	fbRPC:				ASyncRPC;
END_VAR


FunctionType:=FUNCTION_TYPE.FUNCTION_TYPE_ASYNC_RPC;
FunctionNumber:=GANTRY_ASYNC_FUNCTION_NUMBER.GANTRY_ASYNC_FUNCTION_PL;
ParameterDW:=0;
ParameterB:=0;
ParametersOK:=FALSE;

IF En THEN
	IF PickStation<=4 AND PickStation>=1 THEN
		IF PickPosition<=9 AND PickPosition>=1 THEN
			ParametersOK:=TRUE;
			ParameterDW:=INT_TO_DWORD((PickStation*1000+PickPosition*100) + (0*10+0));
		END_IF
	END_IF
END_IF

fbRPC(EN:=En AND ParametersOK, Data:=Data, FunctionType:=FunctionType,FunctionNumber:=FunctionNumber, ParameterDW:=ParameterDW, ParameterB:=ParameterB);

Done:=fbRPC.Done;
Executing:=fbRPC.Executing;
Waiting:=fbRPC.Waiting;
Error:=fbRPC.Error OR (fbRPC.Done AND fbRPC.ReturnValue<0) OR NOT ParametersOK;
Progress:=fbRPC.Progress;

END_FUNCTION_BLOCK

// ---- ComLib/POUs/Public/Level 6 Presentation/Gantry/GantryLeave.TcPOU
{library PUBLIC}
(*  Function to leave a pallet in a specific station and position.  *)
FUNCTION_BLOCK GantryLeave
VAR_INPUT
	En: 				BOOL:=FALSE;			(* Set to true to start *)
	LeaveStation:		StationType;			(* Station number 1-4 *)
	LeavePosition:		PositionType;			(* Position number 1-9 *)
END_VAR
VAR_OUTPUT
	Done: 				BOOL:=FALSE;			(* If true, the command is transmitted ok, to reset set En to false *)
	Executing:			BOOL:=FALSE;			(* True while the command in transmitted *)
	Waiting:			BOOL:=FALSE;			(* True if the command is queued to be transmitted *)
	Error: 				BOOL := FALSE;			(* True if an error occured *)
	Progress:			INT:=0;					(* Function progress *)
END_VAR
VAR_IN_OUT
	Data: 				CommunicationData;		(* Common data structure to connect this function block to a specific Communicator block *)
END_VAR
VAR
	FunctionType: 		FUNCTION_TYPE;
	FunctionNumber: 	INT;
	ParameterDW:	DWORD;
	ParameterB:		BYTE;
	ParametersOK:	BOOL;

	fbRPC:				ASyncRPC;
END_VAR


FunctionType:=FUNCTION_TYPE.FUNCTION_TYPE_ASYNC_RPC;
FunctionNumber:=GANTRY_ASYNC_FUNCTION_NUMBER.GANTRY_ASYNC_FUNCTION_PL;
ParameterDW:=0;
ParameterB:=0;
ParametersOK:=FALSE;

IF En THEN
	IF LeaveStation<=4 AND LeaveStation>=1 THEN
		IF LeavePosition<=9 AND LeavePosition>=1 THEN
			ParametersOK:=TRUE;
			ParameterDW:=INT_TO_DWORD( (0*1000+0*100) + (LeaveStation*10+LeavePosition));
		END_IF
	END_IF
END_IF

fbRPC(EN:=En AND ParametersOK, Data:=Data, FunctionType:=FunctionType,FunctionNumber:=FunctionNumber, ParameterDW:=ParameterDW, ParameterB:=ParameterB);

Done:=fbRPC.Done;
Executing:=fbRPC.Executing;
Waiting:=fbRPC.Waiting;
Error:=fbRPC.Error OR (fbRPC.Done AND fbRPC.ReturnValue<0) OR NOT ParametersOK;
Progress:=fbRPC.Progress;

END_FUNCTION_BLOCK

// ---- ComLib/POUs/Private/_FreeInstance.TcPOU
{library PRIVATE}
(*
  Private Funtcion:
  Frees a previous allocated communications instance.
  Note that it is not possible to free an instance during ongoing read or write (use cancel to break ongoing send or read).

  Return true if station was released. 
*)

FUNCTION _FreeInstance : BOOL
VAR_INPUT
	Instance: 				INT;		(* Instance, a number concatenated by SationNumber (1-INSTANCE_MAX_NUMBER_OF_STATIONS) and DeviceNumber (1-INSTANCE_MAX_NUMBER_OF_DEVICES). Instance is defined as: StaionNumber*100+DeviceNumber *)
END_VAR
VAR
	StationNumber: 		INT;
	StationDevice: 		INT;
END_VAR

_FreeInstance:=FALSE;

IF _CheckInstance(Instance) THEN
	StationNumber:=Instance/100;
	StationDevice:=Instance-StationNumber*100;

	IF ( ComGVL._Instance[StationNumber, StationDevice]<> INSTANCE_STATUS.INSTANCE_STATUS_BUSY) AND
              (ComGVL._Instance[StationNumber, StationDevice]<>INSTANCE_STATUS.INSTANCE_STATUS_CANCEL) THEN

		ComGVL._Instance[StationNumber, StationDevice]:=INSTANCE_STATUS.INSTANCE_STATUS_FREE;
		_FreeInstance:=TRUE;
	END_IF;
END_IF;

END_FUNCTION

// ---- ComLib/POUs/Private/_TryOut.TcPOU
{library PRIVATE}
FUNCTION_BLOCK _TryOut
VAR_INPUT
	Enable: BOOL;
END_VAR
VAR_OUTPUT
END_VAR
VAR
	ABBStatusRestart:		INT:=1;
	
END_VAR

ComGVL._fbTryOutShowABB:=FALSE;
ComGVL._fbTryOutShowGantry:=FALSE;

ComGVL._fbTryOutCommunicator(En:=ComGVL._mxTryOutEnable, Address:=ComGVL._miAddressNumber[ComGVL._miAddressIndex], Data:=ComGVL._msTryOutData);

CASE  ComGVL._glAddressSelectionIndex OF
1,2,3,4:
	ComGVL._fbTryOutShowABB:=TRUE;

	ComGVL._fbTryOutABBGetStatus(En:=ComGVL._fbTryOutABBGoToHomeEn, Data:=ComGVL._msTryOutData);
	IF ComGVL._fbTryOutABBGetStatus.Done THEN
		ComGVL._fbTryOutABBRunMode:=ComGVL._fbTryOutABBGetStatus.RunningMode;
		ComGVL._fbTryOutABBOpMode:=ComGVL._fbTryOutABBGetStatus.OperatingMode;
		ABBStatusRestart:=ABBStatusRestart+1;
		IF ABBStatusRestart=4 THEN
			ABBStatusRestart:=1;
			ComGVL._fbTryOutABBGetStatus(En:=FALSE, Data:=ComGVL._msTryOutData);
		END_IF;
	END_IF;

	(* GoTo *)
	ComGVL._fbTryOutABBGoToHome(En:=ComGVL._fbTryOutABBGoToHomeEn, Data:=ComGVL._msTryOutData);
	IF ComGVL._fbTryOutABBGoToHome.En THEN
		ComGVL._fbTryOutDone:=ComGVL._fbTryOutABBGoToHome.Done;
		ComGVL._fbTryOutExecuting:=ComGVL._fbTryOutABBGoToHome.Executing;
		ComGVL._fbTryOutWaiting:=ComGVL._fbTryOutABBGoToHome.Waiting;
		ComGVL._fbTryOutError:=ComGVL._fbTryOutABBGoToHome.Error;
		ComGVL._fbTryOutProgress:=ComGVL._fbTryOutABBGoToHome.Progress;
	END_IF;
	
	ComGVL._fbTryOutABBGoToSensor(En:=ComGVL._fbTryOutABBGoToSensorEn, Data:=ComGVL._msTryOutData);
	IF ComGVL._fbTryOutABBGoToSensor.En THEN
		ComGVL._fbTryOutDone:=ComGVL._fbTryOutABBGoToSensor.Done;
		ComGVL._fbTryOutExecuting:=ComGVL._fbTryOutABBGoToSensor.Executing;
		ComGVL._fbTryOutWaiting:=ComGVL._fbTryOutABBGoToSensor.Waiting;
		ComGVL._fbTryOutError:=ComGVL._fbTryOutABBGoToSensor.Error;
		ComGVL._fbTryOutProgress:=ComGVL._fbTryOutABBGoToSensor.Progress;
	END_IF;
	
	ComGVL._fbTryOutABBGoToStorage(En:=ComGVL._fbTryOutABBGoToStorageEn, Data:=ComGVL._msTryOutData);
	IF ComGVL._fbTryOutABBGoToStorage.En THEN
		ComGVL._fbTryOutDone:=ComGVL._fbTryOutABBGoToStorage.Done;
		ComGVL._fbTryOutExecuting:=ComGVL._fbTryOutABBGoToStorage.Executing;
		ComGVL._fbTryOutWaiting:=ComGVL._fbTryOutABBGoToStorage.Waiting;
		ComGVL._fbTryOutError:=ComGVL._fbTryOutABBGoToStorage.Error;
		ComGVL._fbTryOutProgress:=ComGVL._fbTryOutABBGoToStorage.Progress;
	END_IF;
	
	ComGVL._fbTryOutABBGoToTable(En:=ComGVL._fbTryOutABBGoToTableEn, Data:=ComGVL._msTryOutData);
	IF ComGVL._fbTryOutABBGoToTable.En THEN
		ComGVL._fbTryOutDone:=ComGVL._fbTryOutABBGoToTable.Done;
		ComGVL._fbTryOutExecuting:=ComGVL._fbTryOutABBGoToTable.Executing;
		ComGVL._fbTryOutWaiting:=ComGVL._fbTryOutABBGoToTable.Waiting;
		ComGVL._fbTryOutError:=ComGVL._fbTryOutABBGoToTable.Error;
		ComGVL._fbTryOutProgress:=ComGVL._fbTryOutABBGoToTable.Progress;
	END_IF;

	ComGVL._fbTryOutABBGoToConveyor1(En:=ComGVL._fbTryOutABBGoToConveyor1En, Data:=ComGVL._msTryOutData);
	IF ComGVL._fbTryOutABBGoToConveyor1.En THEN
		ComGVL._fbTryOutDone:=ComGVL._fbTryOutABBGoToConveyor1.Done;
		ComGVL._fbTryOutExecuting:=ComGVL._fbTryOutABBGoToConveyor1.Executing;
		ComGVL._fbTryOutWaiting:=ComGVL._fbTryOutABBGoToConveyor1.Waiting;
		ComGVL._fbTryOutError:=ComGVL._fbTryOutABBGoToConveyor1.Error;
		ComGVL._fbTryOutProgress:=ComGVL._fbTryOutABBGoToConveyor1.Progress;
	END_IF;
	
	ComGVL._fbTryOutABBGoToConveyor2(En:=ComGVL._fbTryOutABBGoToConveyor2En, Data:=ComGVL._msTryOutData);
	IF ComGVL._fbTryOutABBGoToConveyor2.En THEN
		ComGVL._fbTryOutDone:=ComGVL._fbTryOutABBGoToConveyor2.Done;
		ComGVL._fbTryOutExecuting:=ComGVL._fbTryOutABBGoToConveyor2.Executing;
		ComGVL._fbTryOutWaiting:=ComGVL._fbTryOutABBGoToConveyor2.Waiting;
		ComGVL._fbTryOutError:=ComGVL._fbTryOutABBGoToConveyor2.Error;
		ComGVL._fbTryOutProgress:=ComGVL._fbTryOutABBGoToConveyor2.Progress;
	END_IF;
	
	(* Pick Leave *)
	ComGVL._fbTryOutABBPickLeaveSensor(En:=ComGVL._fbTryOutABBPickLeaveSensorEn, Data:=ComGVL._msTryOutData, Pick:=ComGVL._fbTryOutABBPSensor);
	IF ComGVL._fbTryOutABBPickLeaveSensor.En THEN
		ComGVL._fbTryOutDone:=ComGVL._fbTryOutABBPickLeaveSensor.Done;
		ComGVL._fbTryOutExecuting:=ComGVL._fbTryOutABBPickLeaveSensor.Executing;
		ComGVL._fbTryOutWaiting:=ComGVL._fbTryOutABBPickLeaveSensor.Waiting;
		ComGVL._fbTryOutError:=ComGVL._fbTryOutABBPickLeaveSensor.Error;
		ComGVL._fbTryOutProgress:=ComGVL._fbTryOutABBPickLeaveSensor.Progress;
	END_IF;
	
	ComGVL._fbTryOutABBPickLeaveStorage(En:=ComGVL._fbTryOutABBPickLeaveStorageEn, Data:=ComGVL._msTryOutData, Pick:=ComGVL._fbTryOutABBPStorage, Position:=ComGVL._fbTryOutABBPStoragePos);
	IF ComGVL._fbTryOutABBPickLeaveStorage.En THEN
		ComGVL._fbTryOutDone:=ComGVL._fbTryOutABBPickLeaveStorage.Done;
		ComGVL._fbTryOutExecuting:=ComGVL._fbTryOutABBPickLeaveStorage.Executing;
		ComGVL._fbTryOutWaiting:=ComGVL._fbTryOutABBPickLeaveStorage.Waiting;
		ComGVL._fbTryOutError:=ComGVL._fbTryOutABBPickLeaveStorage.Error;
		ComGVL._fbTryOutProgress:=ComGVL._fbTryOutABBPickLeaveStorage.Progress;
	END_IF;
	
	ComGVL._fbTryOutABBPickLeaveTable(En:=ComGVL._fbTryOutABBPickLeaveTableEn, Data:=ComGVL._msTryOutData, Pick:=ComGVL._fbTryOutABBPTable, Position:=ComGVL._fbTryOutABBPTablePos);
	IF ComGVL._fbTryOutABBPickLeaveTable.En THEN
		ComGVL._fbTryOutDone:=ComGVL._fbTryOutABBPickLeaveTable.Done;
		ComGVL._fbTryOutExecuting:=ComGVL._fbTryOutABBPickLeaveTable.Executing;
		ComGVL._fbTryOutWaiting:=ComGVL._fbTryOutABBPickLeaveTable.Waiting;
		ComGVL._fbTryOutError:=ComGVL._fbTryOutABBPickLeaveTable.Error;
		ComGVL._fbTryOutProgress:=ComGVL._fbTryOutABBPickLeaveTable.Progress;
	END_IF;
	
	ComGVL._fbTryOutABBPickLeaveTable(En:=ComGVL._fbTryOutABBPickLeaveTableEn, Data:=ComGVL._msTryOutData, Pick:=ComGVL._fbTryOutABBPTable, Position:=ComGVL._fbTryOutABBPTablePos);
	IF ComGVL._fbTryOutABBPickLeaveTable.En THEN
		ComGVL._fbTryOutDone:=ComGVL._fbTryOutABBPickLeaveTable.Done;
		ComGVL._fbTryOutExecuting:=ComGVL._fbTryOutABBPickLeaveTable.Executing;
		ComGVL._fbTryOutWaiting:=ComGVL._fbTryOutABBPickLeaveTable.Waiting;
		ComGVL._fbTryOutError:=ComGVL._fbTryOutABBPickLeaveTable.Error;
		ComGVL._fbTryOutProgress:=ComGVL._fbTryOutABBPickLeaveTable.Progress;
	END_IF;
	
	ComGVL._fbTryOutABBPickLeaveConveyor1(En:=ComGVL._fbTryOutABBPickLeaveConveyor1En, Data:=ComGVL._msTryOutData, Pick:=ComGVL._fbTryOutABBPConveyor1);
	IF ComGVL._fbTryOutABBPickLeaveConveyor1.En THEN
		ComGVL._fbTryOutDone:=ComGVL._fbTryOutABBPickLeaveConveyor1.Done;
		ComGVL._fbTryOutExecuting:=ComGVL._fbTryOutABBPickLeaveConveyor1.Executing;
		ComGVL._fbTryOutWaiting:=ComGVL._fbTryOutABBPickLeaveConveyor1.Waiting;
		ComGVL._fbTryOutError:=ComGVL._fbTryOutABBPickLeaveConveyor1.Error;
		ComGVL._fbTryOutProgress:=ComGVL._fbTryOutABBPickLeaveConveyor1.Progress;
	END_IF;
	
	ComGVL._fbTryOutABBPickLeaveConveyor2(En:=ComGVL._fbTryOutABBPickLeaveConveyor2En, Data:=ComGVL._msTryOutData, Pick:=ComGVL._fbTryOutABBPConveyor2);
	IF ComGVL._fbTryOutABBPickLeaveConveyor2.En THEN
		ComGVL._fbTryOutDone:=ComGVL._fbTryOutABBPickLeaveConveyor2.Done;
		ComGVL._fbTryOutExecuting:=ComGVL._fbTryOutABBPickLeaveConveyor2.Executing;
		ComGVL._fbTryOutWaiting:=ComGVL._fbTryOutABBPickLeaveConveyor2.Waiting;
		ComGVL._fbTryOutError:=ComGVL._fbTryOutABBPickLeaveConveyor2.Error;
		ComGVL._fbTryOutProgress:=ComGVL._fbTryOutABBPickLeaveConveyor2.Progress;
	END_IF;

5:
	ComGVL._fbTryOutShowGantry:=TRUE;

	ComGVL._fbTryOutGantryPick(En:=ComGVL._fbTryOutGantryPickEn, Data:=ComGVL._msTryOutData, PickStation:=ComGVL._fbTryOutGantryPickStation, PickPosition:=ComGVL._fbTryOutGantryPickPos);
	IF ComGVL._fbTryOutGantryPick.En THEN
		ComGVL._fbTryOutDone:=ComGVL._fbTryOutGantryPick.Done;
		ComGVL._fbTryOutExecuting:=ComGVL._fbTryOutGantryPick.Executing;
		ComGVL._fbTryOutWaiting:=ComGVL._fbTryOutGantryPick.Waiting;
		ComGVL._fbTryOutError:=ComGVL._fbTryOutGantryPick.Error;
		ComGVL._fbTryOutProgress:=ComGVL._fbTryOutGantryPick.Progress;
	END_IF;

	ComGVL._fbTryOutGantryLeave(En:=ComGVL._fbTryOutGantryLeaveEn, Data:=ComGVL._msTryOutData, LeaveStation:=ComGVL._fbTryOutGantryLeaveStation, LeavePosition:=ComGVL._fbTryOutGantryLeavePos);
	IF ComGVL._fbTryOutGantryLeave.En THEN
		ComGVL._fbTryOutDone:=ComGVL._fbTryOutGantryLeave.Done;
		ComGVL._fbTryOutExecuting:=ComGVL._fbTryOutGantryLeave.Executing;
		ComGVL._fbTryOutWaiting:=ComGVL._fbTryOutGantryLeave.Waiting;
		ComGVL._fbTryOutError:=ComGVL._fbTryOutGantryLeave.Error;
		ComGVL._fbTryOutProgress:=ComGVL._fbTryOutGantryLeave.Progress;
	END_IF;

END_CASE

ComGVL._fbTryOutGetStatus(En:=TRUE, Data:=ComGVL._msTryOutData);
ComGVL._fbTryOutGetStatusRunning:=ComGVL._fbTryOutGetStatus.Running;
ComGVL._fbTryOutGetStatusProgress:=ComGVL._fbTryOutGetStatus.Progress;
ComGVL._fbTryOutGetStatusProgramNumber:=ComGVL._fbTryOutGetStatus.ProgramNumber;
ComGVL._fbTryOutGetStatusHeartBeat:=ComGVL._fbTryOutGetStatus.HeartBeat;
ComGVL._fbTryOutGetStatusError:=ComGVL._fbTryOutGetStatus.Error;

END_FUNCTION_BLOCK

// ---- ComLib/POUs/Public/Level 2 Data link/DeviceClose.TcPOU
{library PUBLIC}
(* Use this function to close an open communication link to a specific device defined by Instance.
Returnvalue is true if closed ok otherwise false.*)
FUNCTION DeviceClose : BOOL
VAR_INPUT
	Instance: 				INT;		(* Instance is an address, use the function ToAddress() to convert station and device number to a valid address. *)
END_VAR

DeviceClose:=FALSE;
IF _GetInstance(Instance)=INSTANCE_STATUS.INSTANCE_STATUS_READY THEN
	IF _FreeInstance(Instance) THEN
		DeviceClose:=TRUE;
	END_IF;
END_IF;

END_FUNCTION

// ---- ComLib/POUs/Public/Level 2 Data link/DeviceStatus.TcPOU
{library PUBLIC}
(* Use this function block toget status of a specific device instance.*)
FUNCTION_BLOCK DeviceStatus
VAR_INPUT
	En:						BOOL;		(* Enable signal, if true this block will give new status values *)
	Instance: 				INT;		(* Instance is an address, use the function ToAddress() to convert station and device number to a valid address. *)
END_VAR
VAR_OUTPUT
	Done:					BOOL:=FALSE;			(* True if status was read  *)
	Status: 				INSTANCE_STATUS;		(* Global status for a specific device *)
END_VAR
VAR
END_VAR

IF En THEN
	Status:=_GetInstance(Instance);
	Done:=TRUE;
ELSE
	Done:=FALSE;
END_IF;

END_FUNCTION_BLOCK

// ---- ComLib/POUs/Public/Level 2 Data link/DeviceUse.TcPOU
{library PUBLIC}
(* Use this function block to handle a communication link to a specific device defined by Instance.*)
FUNCTION_BLOCK DeviceUse
VAR_INPUT
	En:						BOOL;					(* Enable signal, if true this block will try to open the device  for communication use, if false and if device was opened it will be closed (Note: may take some time) *)
	Instance: 				INT;					(* Instance is an address, use the function ToAddress() to convert station and device number to a valid address. *)
END_VAR
VAR_OUTPUT
	Done:					BOOL:=FALSE;		(* True if a device was open (note: will remain false until a device is open), will go to false when a previous open device is closed *)
	Status: 				INSTANCE_STATUS;	(* Global status for a specific device *)
END_VAR
VAR
	OldInstance: INT;
END_VAR

Status:=_GetInstance(Instance);

IF En THEN
	IF Status=INSTANCE_STATUS.INSTANCE_STATUS_FREE THEN
		Done:=DeviceOpen(Instance);
		OldInstance:=Instance;
	END_IF;
ELSE
	IF Done THEN
		IF DeviceClose(OldInstance) THEN
			Done:=FALSE;
		END_IF;
	END_IF;
END_IF;

END_FUNCTION_BLOCK

// ---- ComLib/POUs/Public/Level 5 Session/RPC Remote Procedural Call/ASyncProgress.TcPOU
{library PUBLIC}
(*
Get progress value for ASync calls.
This function block will read the global status.
To see a specific function progress use the output of RPCx or ASyncRP function blocks.
*)

FUNCTION_BLOCK ASyncProgress
VAR_INPUT
	En: 				BOOL;			(* Set to true to get progress value *)
END_VAR
VAR_OUTPUT
	Done:				BOOL;			(* Done = En *)
	Progress: 			INT;			(* Progress value *)
END_VAR
VAR_IN_OUT
	Data: 				CommunicationData;		(* Common data structure to connect this function block to a specific Communicator block *)
END_VAR
VAR
END_VAR

IF En THEN
	Progress:=Data._ASyncProgress;
ELSE
	Progress:=0;
END_IF;

Done:=En;

END_FUNCTION_BLOCK

// ---- ComLib/POUs/Public/Level 5 Session/RPC Remote Procedural Call/RPC2.TcPOU
{library PUBLIC}
(*
RPC2 will handle RPC calls with 2 parameters.
A session will be established to the specific equipment during the function call and when a return value exist (or error) the session is ended.
Note, if FunctionType is set to ASync, RPC will only start a function and not wait for the function to end.

It is possible to queue many calls by cascade coupled blocks in serie or parallel.
By using the Done output signal as input to En on another function blockit is possible to serialise calls.

*)
FUNCTION_BLOCK RPC2
VAR_INPUT
	En: 				BOOL:=FALSE;			(* Set to true to call a  RPC 1 parameter function *)
	FunctionType1:	FUNCTION_TYPE:=FUNCTION_TYPE.FUNCTION_TYPE_SYNC_RPC;		(* Function type 1 must be of type SYNC *)
	FunctionNumber1:INT;						(* RPC function number 1 *)
	ParameterDW1:	DWORD;					(* DWORD parameter value 1 *)
	ParameterB1:		BYTE;						(* Byte parameter value 1 *)
	FunctionType2:	FUNCTION_TYPE:=FUNCTION_TYPE.FUNCTION_TYPE_SYNC_RPC;		(*Function type 2 must be of type SYNC *)
	FunctionNumber2:INT;						(* RPC function number 2 *)
	ParameterDW2:	DWORD;					(* DWORD parameter value 2 *)
	ParameterB2:		BYTE;						(* Byte parameter value 2 *)
END_VAR
VAR_OUTPUT
	Done: 				BOOL:=FALSE;			(* If true, the command is transmitted ok, to reset set En to false *)
	Executing:			BOOL:=FALSE;			(* True while the command in transmitted *)
	Waiting:			BOOL:=FALSE;			(* True if the command is queued to be transmitted *)
	Error: 				BOOL := FALSE;			(* True if an communication error occured *)
	ReturnValue1:		FUNCTION_TYPE;		(* Return value *)
	ReturnValue2:		DWORD;					(* DWORD return value *)
	ReturnValue3:		BYTE;						(* BYTE return value *)
END_VAR
VAR_IN_OUT
	Data: 				CommunicationData;		(* Common data structure to connect this function block to a specific Communicator block *)
END_VAR
VAR
	fbSessionInit: 		SessionInit;
	fbSessionSend1: 	SessionSend;
	fbSessionSend2: 	SessionSend;
	fbSessionEnd: 	SessionEnd;
	Memory: 			BOOL := FALSE;
END_VAR

fbSessionInit(En:=En, Data:=Data);
fbSessionSend1(En:=fbSessionInit.Done, SessionID:=fbSessionInit.SessionID, Data:=Data,
					FunctionType:=INT_TO_BYTE(FunctionType1), FunctionNumber:=INT_TO_BYTE(FunctionNumber1),
 					ParameterDW:=ParameterDW1, ParameterB:=ParameterB1);

fbSessionSend2(En:=fbSessionInit.Done, SessionID:=fbSessionInit.SessionID, Data:=Data,
					FunctionType:=INT_TO_BYTE(FunctionType2), FunctionNumber:=INT_TO_BYTE(FunctionNumber2),
					ParameterDW:=ParameterDW2, ParameterB:=ParameterB2);

fbSessionEnd(En:=fbSessionSend2.Done, Data:=Data);

Done:=fbSessionSend2.Done;
Executing:=fbSessionSend1.Executing OR fbSessionSend1.Executing;
Waiting:=fbSessionSend1.Waiting;
Error:=fbSessionSend1.Error OR fbSessionSend2.Error;


IF fbSessionSend2.Done AND NOT Memory THEN
	Memory:=TRUE;
	ReturnValue1:=fbSessionSend2.Answer.FunctionType;
	ReturnValue2:=fbSessionSend2.Answer.ParameterDW;
	ReturnValue3:=fbSessionSend2.Answer.ParameterB;
ELSIF NOT En THEN
	ReturnValue1:=FUNCTION_TYPE.FUNCTION_TYPE_ERROR_NO_FUNCTION;
	Memory:=FALSE;
ELSE
	Memory:=FALSE;
	ReturnValue1:=FUNCTION_TYPE.FUNCTION_TYPE_ERROR_BUSY;
END_IF;

END_FUNCTION_BLOCK

// ---- ComLib/POUs/Public/Level 6 Presentation/ABB/IO/ABBIORead.TcPOU
{library PUBLIC}
(* Function to read a DI I/O *)
FUNCTION_BLOCK ABBIORead
VAR_INPUT
	En: 			BOOL:=FALSE;				(* Set to true to start *)
	IONumber:		INT:=0;						(* DI I/O number to read *)
END_VAR
VAR_OUTPUT
	Done: 				BOOL:=FALSE;			(* If true, the command is transmitted ok, to reset set En to false *)
	Executing:			BOOL:=FALSE;			(* True while the command in transmitted *)
	Waiting:			BOOL:=FALSE;			(* True if the command is queued to be transmitted *)
	Error: 				BOOL := FALSE;			(* True if an error occured *)
	Progress:			INT:=0;					(* Function progress *)
	Value:				BOOL:=FALSE;			(* I/O return value *)
END_VAR
VAR_IN_OUT
	Data: 				CommunicationData;		(* Common data structure to connect this function block to a specific Communicator block *)
END_VAR
VAR
	FunctionType: 		FUNCTION_TYPE;
	FunctionNumber: 	INT;
	ParameterDW:		DWORD;
	ParameterB:			BYTE;
	Sequence:			INT:=0;

	fbRPC:				RPC1;
END_VAR

FunctionType:=FUNCTION_TYPE.FUNCTION_TYPE_SYNC_RPC;
FunctionNumber:=ABB_SYNC_FUNCTION_NUMBER.ABB_SYNC_READ_DI;
ParameterDW:=INT_TO_DWORD(IONumber);

fbRPC(EN:=En, Data:=Data, FunctionType1:=FunctionType,FunctionNumber1:=FunctionNumber, ParameterDW1:=ParameterDW, ParameterB1:=ParameterB);

Done:=fbRPC.Done;
Executing:=fbRPC.Executing;
Waiting:=fbRPC.Waiting;
Error:=fbRPC.Error;
Progress:=100*BOOL_TO_INT(Done);
Value:=BYTE_TO_BOOL(fbRPC.ReturnValue3);

END_FUNCTION_BLOCK

// ---- ComLib/POUs/Public/Level 6 Presentation/ABB/IO/ABBIOReadValve.TcPOU
{library PUBLIC}
(* Function to read a valve value (open or closed) *)
FUNCTION_BLOCK ABBIOReadValve
VAR_INPUT
	En: 			BOOL:=FALSE;				(* Set to true to start *)
	Valve:			INT:=0;						(* Valve I/O number *)
END_VAR
VAR_OUTPUT
	Done: 				BOOL:=FALSE;			(* If true, the command is transmitted ok, to reset set En to false *)
	Executing:			BOOL:=FALSE;			(* True while the command in transmitted *)
	Waiting:			BOOL:=FALSE;			(* True if the command is queued to be transmitted *)
	Error: 				BOOL := FALSE;			(* True if an error occured *)
	Progress:			INT:=0;					(* Function progress *)
	Value:				BOOL:=FALSE;			(* FALSE=open, TRUE=closed *)
END_VAR
VAR_IN_OUT
	Data: 				CommunicationData;		(* Common data structure to connect this function block to a specific Communicator block *)
END_VAR
VAR
	FunctionType: 		FUNCTION_TYPE;
	FunctionNumber: 	INT;
	ParameterDW:	DWORD;
	ParameterB:		BYTE;
	Sequence:			INT:=0;

	fbRPC:				RPC1;
END_VAR

FunctionType:=FUNCTION_TYPE.FUNCTION_TYPE_SYNC_RPC;
FunctionNumber:=ABB_SYNC_FUNCTION_NUMBER.ABB_SYNC_WRITE_DO;
ParameterDW:=INT_TO_DWORD(Valve);
ParameterB:=0;

fbRPC(EN:=En, Data:=Data, FunctionType1:=FunctionType,FunctionNumber1:=FunctionNumber, ParameterDW1:=ParameterDW, ParameterB1:=ParameterB);

Done:=fbRPC.Done;
Executing:=fbRPC.Executing;
Waiting:=fbRPC.Waiting;
Error:=fbRPC.Error;
Progress:=100*BOOL_TO_INT(Done);
Value:=BYTE_TO_BOOL(fbRPC.ReturnValue3);

END_FUNCTION_BLOCK

// ---- ComLib/POUs/Public/Level 6 Presentation/ABB/IO/ABBIOWrite.TcPOU
{library PUBLIC}
(* Function to write a DO I/O *)
FUNCTION_BLOCK ABBIOWrite
VAR_INPUT
	En: 			BOOL:=FALSE;				(* Set to true to start *)
	IONumber:		INT:=0;						(* DO I/O number to read *)
END_VAR
VAR_OUTPUT
	Done: 				BOOL:=FALSE;			(* If true, the command is transmitted ok, to reset set En to false *)
	Executing:			BOOL:=FALSE;			(* True while the command in transmitted *)
	Waiting:			BOOL:=FALSE;			(* True if the command is queued to be transmitted *)
	Error: 				BOOL := FALSE;			(* True if an error occured *)
	Progress:			INT:=0;					(* Function progress *)
END_VAR
VAR_IN_OUT
	Data: 				CommunicationData;		(* Common data structure to connect this function block to a specific Communicator block *)
END_VAR
VAR
	FunctionType: 		FUNCTION_TYPE;
	FunctionNumber: 	INT;
	ParameterDW:	DWORD;
	ParameterB:		BYTE;
	Sequence:			INT:=0;

	fbRPC:				RPC1;
END_VAR

FunctionType:=FUNCTION_TYPE.FUNCTION_TYPE_SYNC_RPC;
FunctionNumber:=ABB_SYNC_FUNCTION_NUMBER.ABB_SYNC_WRITE_DO;
ParameterDW:=INT_TO_DWORD(IONumber);

fbRPC(EN:=En, Data:=Data, FunctionType1:=FunctionType,FunctionNumber1:=FunctionNumber, ParameterDW1:=ParameterDW, ParameterB1:=ParameterB);

Done:=fbRPC.Done;
Executing:=fbRPC.Executing;
Waiting:=fbRPC.Waiting;
Error:=fbRPC.Error;
Progress:=100*BOOL_TO_INT(Done);

END_FUNCTION_BLOCK

// ---- ComLib/POUs/Public/Level 6 Presentation/ABB/IO/ABBIOWriteValve.TcPOU
{library PUBLIC}
(* Function to write a value to valve I/O *)
FUNCTION_BLOCK ABBIOWriteValve
VAR_INPUT
	En: 			BOOL:=FALSE;				(* Set to true to start *)
	Valve:			INT:=0;							(* Valve I/O number *)
	Value:			BOOL:=FALSE;				(* FALSE=open, TRUE=closed *)
END_VAR
VAR_OUTPUT
	Done: 				BOOL:=FALSE;			(* If true, the command is transmitted ok, to reset set En to false *)
	Executing:			BOOL:=FALSE;			(* True while the command in transmitted *)
	Waiting:			BOOL:=FALSE;			(* True if the command is queued to be transmitted *)
	Error: 				BOOL := FALSE;			(* True if an error occured *)
	Progress:			INT:=0;					(* Function progress *)
END_VAR
VAR_IN_OUT
	Data: 				CommunicationData;		(* Common data structure to connect this function block to a specific Communicator block *)
END_VAR
VAR
	FunctionType: 		FUNCTION_TYPE;
	FunctionNumber: 	INT;
	ParameterDW:	DWORD;
	ParameterB:		BYTE;
	Sequence:			INT:=0;

	fbRPC:				RPC1;
END_VAR

FunctionType:=FUNCTION_TYPE.FUNCTION_TYPE_SYNC_RPC;
FunctionNumber:=ABB_SYNC_FUNCTION_NUMBER.ABB_SYNC_WRITE_DO;
ParameterDW:=INT_TO_DWORD(Valve);
ParameterB:=BOOL_TO_BYTE(Value);

fbRPC(EN:=En, Data:=Data, FunctionType1:=FunctionType,FunctionNumber1:=FunctionNumber, ParameterDW1:=ParameterDW, ParameterB1:=ParameterB);

Done:=fbRPC.Done;
Executing:=fbRPC.Executing;
Waiting:=fbRPC.Waiting;
Error:=fbRPC.Error;
Progress:=100*BOOL_TO_INT(Done);

END_FUNCTION_BLOCK

// ---- ComLib/POUs/Public/Level 6 Presentation/ABB/Move/ABBMoveJAbs.TcPOU
{library PUBLIC}
(* Function to move a robot to an abs location *)
FUNCTION_BLOCK ABBMoveJAbs
VAR_INPUT
	En: 				BOOL:=FALSE;			(* Set to true to start *)
	X:					REAL:=0.0;				(* X position *)
	Y:					REAL:=0.0;				(* Y position *)
	Z:					REAL:=0.0;				(* Z position *)
	RX:					REAL:=0.0;				(* RX angle *)
	RY:					REAL:=0.0;				(* RY angle *)
	RZ:					REAL:=0.0;				(* RZ angle *)
END_VAR
VAR_OUTPUT
	Done: 				BOOL:=FALSE;			(* If true, the command is transmitted ok, to reset set En to false *)
	Executing:			BOOL:=FALSE;			(* True while the command in transmitted *)
	Waiting:			BOOL:=FALSE;			(* True if the command is queued to be transmitted *)
	Error: 				BOOL := FALSE;			(* True if an error occured *)
	Progress:			INT:=0;					(* Function progress *)
END_VAR
VAR_IN_OUT
	Data: 				CommunicationData;		(* Common data structure to connect this function block to a specific Communicator block *)
END_VAR
VAR
	FunctionType: 		FUNCTION_TYPE;
	FunctionNumber: 	INT;
	ParameterDW:	DWORD;
	ParameterB:		BYTE;
	Sequence:			INT:=0;

	fbRPC:				ASyncRPC;
END_VAR

FunctionType:=FUNCTION_TYPE.FUNCTION_TYPE_ASYNC_RPC;
FunctionNumber:=ABB_ASYNC_ABS_MOVEJ_TO_POSE;
ParameterDW:=0;										(* No parameters *)
ParameterB:=0;

fbRPC(EN:=En, Data:=Data, FunctionType:=FunctionType,FunctionNumber:=FunctionNumber, ParameterDW:=ParameterDW, ParameterB:=ParameterB);

Done:=fbRPC.Done;
Executing:=fbRPC.Executing;
Waiting:=fbRPC.Waiting;
Error:=fbRPC.Error OR (fbRPC.Done AND fbRPC.ReturnValue<0);
Progress:=fbRPC.Progress;

END_FUNCTION_BLOCK

// ---- ComLib/POUs/Public/Level 6 Presentation/ABB/Move/ABBMoveJRel.TcPOU
{library PUBLIC}
(* Function to move a robot relative current location *)
FUNCTION_BLOCK ABBMoveJRel
VAR_INPUT
	En: 				BOOL:=FALSE;			(* Set to true to start *)
	X:					REAL:=0.0;				(* X position *)
	Y:					REAL:=0.0;				(* Y position *)
	Z:					REAL:=0.0;				(* Z position *)
	RX:					REAL:=0.0;				(* RX angle *)
	RY:					REAL:=0.0;				(* RY angle *)
	RZ:					REAL:=0.0;				(* RZ angle *)
END_VAR
VAR_OUTPUT
	Done: 				BOOL:=FALSE;			(* If true, the command is transmitted ok, to reset set En to false *)
	Executing:			BOOL:=FALSE;			(* True while the command in transmitted *)
	Waiting:			BOOL:=FALSE;			(* True if the command is queued to be transmitted *)
	Error: 				BOOL := FALSE;			(* True if an error occured *)
	Progress:			INT:=0;						(* Function progress *)
END_VAR
VAR_IN_OUT
	Data: 				CommunicationData;		(* Common data structure to connect this function block to a specific Communicator block *)
END_VAR
VAR
	FunctionType: 		FUNCTION_TYPE;
	FunctionNumber: 	INT;
	ParameterDW:	DWORD;
	ParameterB:		BYTE;
	Sequence:			INT:=0;

	fbRPC:				ASyncRPC;
END_VAR

FunctionType:=FUNCTION_TYPE.FUNCTION_TYPE_ASYNC_RPC;
FunctionNumber:=ABB_ASYNC_REL_MOVEJ_TO_POSE;
ParameterDW:=0;										(* No parameters *)
ParameterB:=0;

fbRPC(EN:=En, Data:=Data, FunctionType:=FunctionType,FunctionNumber:=FunctionNumber, ParameterDW:=ParameterDW, ParameterB:=ParameterB);

Done:=fbRPC.Done;
Executing:=fbRPC.Executing;
Waiting:=fbRPC.Waiting;
Error:=fbRPC.Error OR (fbRPC.Done AND fbRPC.ReturnValue<0);
Progress:=fbRPC.Progress;

END_FUNCTION_BLOCK

// ---- ComLib/POUs/Public/Level 6 Presentation/ABB/Move/ABBMoveLAbs.TcPOU
{library PUBLIC}
(* Function to move a robot to an abs location *)
FUNCTION_BLOCK ABBMoveLAbs
VAR_INPUT
	En: 				BOOL:=FALSE;			(* Set to true to start *)
	X:					REAL:=0.0;				(* X position *)
	Y:					REAL:=0.0;				(* Y position *)
	Z:					REAL:=0.0;				(* Z position *)
	RX:					REAL:=0.0;				(* RX angle *)
	RY:					REAL:=0.0;				(* RY angle *)
	RZ:					REAL:=0.0;				(* RZ angle *)
END_VAR
VAR_OUTPUT
	Done: 				BOOL:=FALSE;			(* If true, the command is transmitted ok, to reset set En to false *)
	Executing:			BOOL:=FALSE;			(* True while the command in transmitted *)
	Waiting:			BOOL:=FALSE;			(* True if the command is queued to be transmitted *)
	Error: 				BOOL := FALSE;			(* True if an error occured *)
	Progress:			INT:=0;						(* Function progress *)
END_VAR
VAR_IN_OUT
	Data: 				CommunicationData;		(* Common data structure to connect this function block to a specific Communicator block *)
END_VAR
VAR
	FunctionType: 		FUNCTION_TYPE;
	FunctionNumber: 	INT;
	ParameterDW:	DWORD;
	ParameterB:		BYTE;
	Sequence:			INT:=0;

	fbRPC:				ASyncRPC;
END_VAR

FunctionType:=FUNCTION_TYPE.FUNCTION_TYPE_ASYNC_RPC;
FunctionNumber:=ABB_ASYNC_ABS_MOVEL_TO_POSE;
ParameterDW:=0;										(* No parameters *)
ParameterB:=0;

fbRPC(EN:=En, Data:=Data, FunctionType:=FunctionType,FunctionNumber:=FunctionNumber, ParameterDW:=ParameterDW, ParameterB:=ParameterB);

Done:=fbRPC.Done;
Executing:=fbRPC.Executing;
Waiting:=fbRPC.Waiting;
Error:=fbRPC.Error OR (fbRPC.Done AND fbRPC.ReturnValue<0);
Progress:=fbRPC.Progress;

END_FUNCTION_BLOCK

// ---- ComLib/POUs/Public/Level 6 Presentation/ABB/Move/ABBMoveLRel.TcPOU
{library PUBLIC}
(* Function to move a robot relative current location *)
FUNCTION_BLOCK ABBMoveLRel
VAR_INPUT
	En: 				BOOL:=FALSE;			(* Set to true to start *)
	X:					REAL:=0.0;				(* X position *)
	Y:					REAL:=0.0;				(* Y position *)
	Z:					REAL:=0.0;				(* Z position *)
	RX:					REAL:=0.0;				(* RX angle *)
	RY:					REAL:=0.0;				(* RY angle *)
	RZ:					REAL:=0.0;				(* RZ angle *)
END_VAR
VAR_OUTPUT
	Done: 				BOOL:=FALSE;			(* If true, the command is transmitted ok, to reset set En to false *)
	Executing:			BOOL:=FALSE;			(* True while the command in transmitted *)
	Waiting:			BOOL:=FALSE;			(* True if the command is queued to be transmitted *)
	Error: 				BOOL := FALSE;			(* True if an error occured *)
	Progress:			INT:=0;						(* Function progress *)
END_VAR
VAR_IN_OUT
	Data: 				CommunicationData;		(* Common data structure to connect this function block to a specific Communicator block *)
END_VAR
VAR
	FunctionType: 		FUNCTION_TYPE;
	FunctionNumber: 	INT;
	ParameterDW:	DWORD;
	ParameterB:		BYTE;
	Sequence:			INT:=0;

	fbRPC:				ASyncRPC;
END_VAR

FunctionType:=FUNCTION_TYPE.FUNCTION_TYPE_ASYNC_RPC;
FunctionNumber:=ABB_ASYNC_REL_MOVEL_TO_POSE;
ParameterDW:=0;										(* No parameters *)
ParameterB:=0;

fbRPC(EN:=En, Data:=Data, FunctionType:=FunctionType,FunctionNumber:=FunctionNumber, ParameterDW:=ParameterDW, ParameterB:=ParameterB);

Done:=fbRPC.Done;
Executing:=fbRPC.Executing;
Waiting:=fbRPC.Waiting;
Error:=fbRPC.Error OR (fbRPC.Done AND fbRPC.ReturnValue<0);
Progress:=fbRPC.Progress;

END_FUNCTION_BLOCK

// ---- ComLib/POUs/Public/Level 6 Presentation/ABB/Pick Leave/ABBProcessAssembly.TcPOU
{library PUBLIC}
(* Function to start a assembly process on the table. *)
FUNCTION_BLOCK ABBProcessAssembly
VAR_INPUT
	En: 				BOOL:=FALSE;			(* Set to true to start *)
END_VAR
VAR_OUTPUT
	Done: 				BOOL:=FALSE;			(* If true, the command is transmitted ok, to reset set En to false *)
	Executing:			BOOL:=FALSE;			(* True while the command in transmitted *)
	Waiting:			BOOL:=FALSE;			(* True if the command is queued to be transmitted *)
	Error: 				BOOL := FALSE;			(* True if an error occured *)
	Progress:			INT:=0;						(* Function progress *)
END_VAR
VAR_IN_OUT
	Data: 				CommunicationData;		(* Common data structure to connect this function block to a specific Communicator block *)
END_VAR
VAR
	FunctionType: 		FUNCTION_TYPE;
	FunctionNumber: 	INT;
	ParameterDW:	DWORD;
	ParameterB:		BYTE;
	Sequence:			INT:=0;

	fbRPC:				ASyncRPC;
END_VAR

FunctionType:=FUNCTION_TYPE.FUNCTION_TYPE_ASYNC_RPC;
FunctionNumber:=ABB_ASYNC_FUNCTION_PROCESS_ASSEMBLY;
ParameterDW:=0;
ParameterB:=0;

fbRPC(EN:=En, Data:=Data, FunctionType:=FunctionType,FunctionNumber:=FunctionNumber, ParameterDW:=ParameterDW, ParameterB:=ParameterB);

Done:=fbRPC.Done;
Executing:=fbRPC.Executing;
Waiting:=fbRPC.Waiting;
Error:=fbRPC.Error OR (fbRPC.Done AND fbRPC.ReturnValue<0);
Progress:=fbRPC.Progress;

END_FUNCTION_BLOCK

// ---- ComLib/POUs/Public/Level 6 Presentation/Gantry/GantryStatus.TcPOU
{library PUBLIC}
(* Function to get gantry status.
    This function can run continuously and will not block other communications.   
 *)
FUNCTION_BLOCK GantryStatus
VAR_INPUT
	En: 					BOOL:=FALSE;			(* Set to true to ask for status, the block  will continuously ask for status while true *)
END_VAR
VAR_OUTPUT
	Done: 					BOOL:=FALSE;			(* If true, the STATUS command is running, to stop/pause set En to false *)
	Status:					GANTRY_STATUS;			(* Gantry status *)
END_VAR
VAR_IN_OUT
	Data: 					CommunicationData;		(* Common data structure to connect this function block to a specific Communicator block *)
END_VAR
VAR
END_VAR


IF En THEN
	
	Status:=NodeReadWord(Address:=Data._Address, Channel:=2);
	Done:=TRUE;
ELSE
	Status:=GANTRY_STATUS.GANTRY_STATUS_NOT_ENABLED;
	Done:=FALSE;
END_IF;

END_FUNCTION_BLOCK

// ---- ComLib/VISUs/Object/_VisuABBGoTo.TcVIS
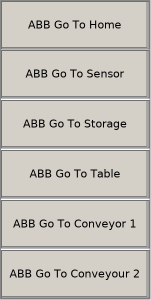
VISUALIZATION _VisuABBGoTo  // 151x300
    Button (1,1 148x48), "ABB Go To Home"
        toggle ComGVL._fbTryOutABBGoToHomeEn
    Button (1,50 148x48), "ABB Go To Sensor"
        toggle ComGVL._fbTryOutABBGoToSensorEn
    Button (1,100 148x48), "ABB Go To Storage"
        toggle ComGVL._fbTryOutABBGoToStorageEn
    Button (1,150 148x48), "ABB Go To Table"
        toggle ComGVL._fbTryOutABBGoToTableEn
    Button (1,200 148x48), "ABB Go To Conveyor 1"
        toggle ComGVL._fbTryOutABBGoToConveyor1En
    Button (1,250 148x48), "ABB Go To Conveyour 2"
        toggle ComGVL._fbTryOutABBGoToConveyor2En
END_VISUALIZATION

// ---- ComLib/VISUs/Object/_VisuABBPickLeave.TcVIS
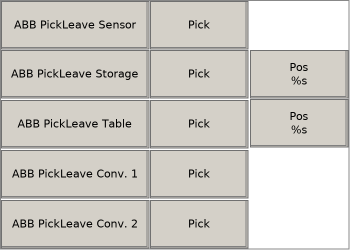
VISUALIZATION _VisuABBPickLeave  // 350x250
    Button (1,1 148x48), "ABB PickLeave Sensor"
        toggle ComGVL._fbTryOutABBPickLeaveSensorEn
    Button (1,50 148x48), "ABB PickLeave Storage"
        toggle ComGVL._fbTryOutABBPickLeaveStorageEn
    Button (1,100 148x48), "ABB PickLeave Table"
        toggle ComGVL._fbTryOutABBPickLeaveTableEn
    Button (1,150 148x48), "ABB PickLeave Conv. 1"
        toggle ComGVL._fbTryOutABBPickLeaveConveyor1En
    Button (1,200 148x48), "ABB PickLeave Conv. 2"
        toggle ComGVL._fbTryOutABBPickLeaveConveyor2En
    Button (150,1 98x48), "Pick"
        toggle ComGVL._fbTryOutABBPSensor
    Button (150,50 98x48), "Pick"
        toggle ComGVL._fbTryOutABBPStorage
    Button (150,100 98x48), "Pick"
        toggle ComGVL._fbTryOutABBPTable
    Button (150,150 98x48), "Pick"
        toggle ComGVL._fbTryOutABBPConveyor1
    Button (150,200 98x48), "Pick"
        toggle ComGVL._fbTryOutABBPConveyor2
    Button (250,50 98x48), "Pos %s", text variable: ComGVL._fbTryOutABBPStoragePos
        OnMouseClick: write the text variable via VisuDialogs.Numpad, min 1, max 9, title 'Position'
    Button (250,99 98x48), "Pos %s", text variable: ComGVL._fbTryOutABBPTablePos
        OnMouseClick: write the text variable via VisuDialogs.Numpad, min 1, max 9, title 'Position'
END_VISUALIZATION

// ---- ComLib/VISUs/Object/_VisuABBStatus.TcVIS
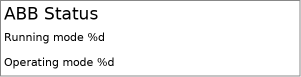
VISUALIZATION _VisuABBStatus  // 301x77
    Label (1,1 148x25), "ABB Status"
    Rectangle (1,25 298x25), "Running mode %d", text variable: ComGVL._gABBRunTable[ComGVL._fbTryOutABBRunMode ]
    Rectangle (1,50 298x25), "Operating mode %d", text variable: ComGVL._gABBOpTable[ComGVL._fbTryOutABBOpMode ]
END_VISUALIZATION

// ---- ComLib/VISUs/Object/_VisuAddressSelector.TcVIS
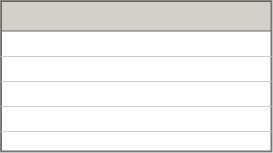
VISUALIZATION _VisuAddressSelector  // 273x153
    Table (1,1 270x150), data array: ComGVL._glAddressNameTable
        p3854506369: ComGVL._glAddressNameTable[INDEX]
        p2232123230: Station Address
        p1137915858: ComGVL._glAddressSelectionIndex
END_VISUALIZATION

// ---- ComLib/VISUs/Object/_VisuAddressShow.TcVIS
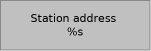
VISUALIZATION _VisuAddressShow  // 151x51
    Rectangle (1,1 148x48), "Station address %s", text variable: ComGVL._glAddressNameTable[ComGVL._glAddressSelectionIndex]
END_VISUALIZATION

// ---- ComLib/VISUs/Object/_VisuCommunicator.TcVIS
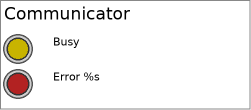
VISUALIZATION _VisuCommunicator  // 251x110
    Lamp1 (1,25 34x48), variable: ComGVL._fbTryOutCommunicator.Busy, style: Lamp-Lamp1-Yellow
    Rectangle (50,25 100x34), "Busy"
    Label (1,1 248x25), "Communicator"
    Lamp1 (1,60 34x48), variable: ComGVL._fbTryOutCommunicator.Error, style: Lamp-Lamp1-Red
    Rectangle (50,60 100x34), "Error %s", text variable: ComGVL._glErrorTable[ComGVL._fbTryOutCommunicator.ErrorID]
END_VISUALIZATION

// ---- ComLib/VISUs/Object/_VisuFunctionCall.TcVIS
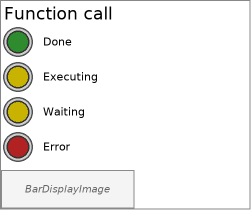
VISUALIZATION _VisuFunctionCall  // 251x210
    Label (1,1 248x25), "Function call"
    Lamp1 (1,25 34x34), variable: ComGVL._fbTryOutDone, style: Lamp-Lamp1-Green
    Lamp1 (1,60 34x34), variable: ComGVL._fbTryOutExecuting, style: Lamp-Lamp1-Yellow
    Lamp1 (1,95 34x34), variable: ComGVL._fbTryOutWaiting, style: Lamp-Lamp1-Yellow
    Lamp1 (1,130 34x34), variable: ComGVL._fbTryOutError, style: Lamp-Lamp1-Red
    BarDisplayImage (1,170 133x38), value: ComGVL._fbTryOutProgress, style: BarDisplayImage-Gray, scale format: %.1f, scale 0..100
    Label (40,25 100x34), "Done"
    Label (40,60 100x34), "Executing"
    Label (40,95 100x34), "Waiting"
    Label (40,130 100x34), "Error"
END_VISUALIZATION

// ---- ComLib/VISUs/Object/_VisuGantryPickLeave.TcVIS
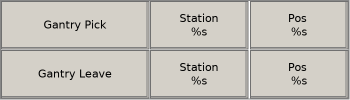
VISUALIZATION _VisuGantryPickLeave  // 350x100
    Button (1,1 148x48), "Gantry Pick"
        toggle ComGVL._fbTryOutGantryPickEn
    Button (1,50 148x48), "Gantry Leave"
        toggle ComGVL._fbTryOutGantryLeaveEn
    Button (150,1 98x48), "Station %s", text variable: ComGVL._fbTryOutGantryPickStation
        OnMouseDown: write the text variable via VisuDialogs.Numpad, min 1, max 4, title 'Station'
    Button (150,50 98x48), "Station %s", text variable: ComGVL._fbTryOutGantryLeaveStation
        OnMouseDown: write the text variable via VisuDialogs.Numpad, min 1, max 4, title 'Station'
    Button (250,1 98x48), "Pos %s", text variable: ComGVL._fbTryOutGantryPickPos
        OnMouseDown: write the text variable via VisuDialogs.Numpad, min 1, max 9, title 'Position'
    Button (250,50 98x48), "Pos %s", text variable: ComGVL._fbTryOutGantryLeavePos
        OnMouseDown: write the text variable via VisuDialogs.Numpad, min 1, max 9, title 'Position'
END_VISUALIZATION

// ---- ComLib/VISUs/Object/_VisuRPCStatusShow.TcVIS
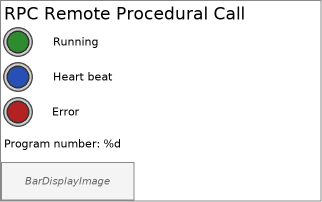
VISUALIZATION _VisuRPCStatusShow  // 322x202
    Lamp1 (1,25 34x34), variable: ComGVL._fbTryOutGetStatusRunning, style: Lamp-Lamp1-Green
    Rectangle (50,25 100x34), "Running"
    Label (1,1 319x25), "RPC Remote Procedural Call"
    Lamp1 (1,60 34x34), variable: ComGVL._fbTryOutGetStatusError, style: Lamp-Lamp1-Blue
    Rectangle (50,60 100x34), "Heart beat"
    Lamp1 (1,95 34x34), variable: ComGVL._fbTryOutGetStatusError, style: Lamp-Lamp1-Red
    Rectangle (49,95 100x34), "Error"
    BarDisplayImage (1,162 133x38), value: ComGVL._fbTryOutGetStatusProgress, style: BarDisplayImage-Gray, scale format: %.1f, scale 0..100
    Rectangle (1,130 176x28), "Program number: %d", text variable: ComGVL._fbTryOutGetStatusProgramNumber
END_VISUALIZATION

// ---- ComLib/VISUs/_TryOut.TcVIS
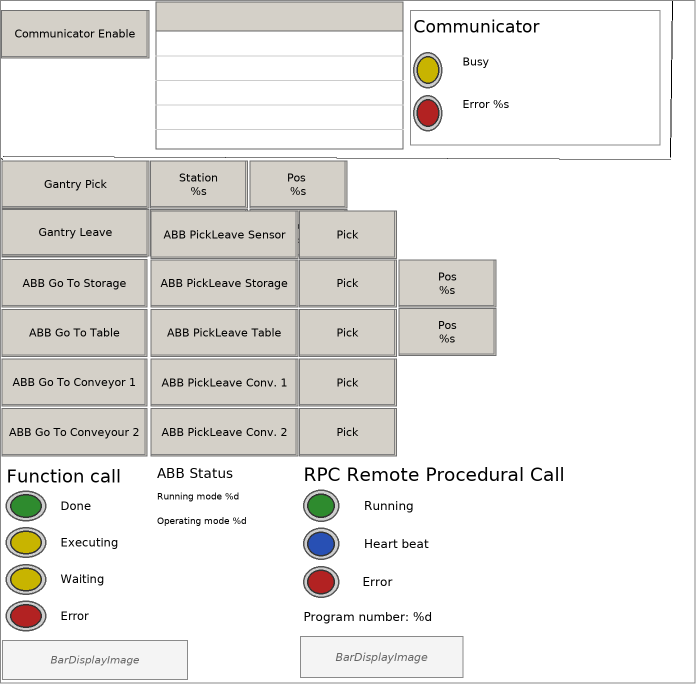
VISUALIZATION _TryOut  // 696x684
    Frame (1,160 148x298), invisible if: not ComGVL._fbTryOutShowABB
        shows _VisuABBGoTo()
    Button (1,10 148x48), "Communicator Enable"
    Frame (155,1 250x150), invisible if: ComGVL._mxTryOutEnable
        shows _VisuAddressSelector()
    Frame (1,160 348x98), invisible if: NOT ComGVL._fbTryOutShowGantry
        shows _VisuGantryPickLeave()
    Frame (150,210 348x248), invisible if: NOT ComGVL._fbTryOutShowABB
        shows _VisuABBPickLeave()
    Frame (154,460 242x75)
        shows _VisuABBStatus()
    Frame (1,462 350x220)
        shows _VisuFunctionCall()
    Frame (410,10 250x135)
        shows _VisuCommunicator()
    Line (1,158) (2,159)
    Line (3,156) (670,159)
    Line (672,1) (670,157)
    Frame (299,460 395x220)
        shows _VisuRPCStatusShow()
END_VISUALIZATION

// ---- GlobalTextList.TcGTLO
TEXTLIST GlobalTextList
  604 = 'ABB Go To Conveyor 1'
  605 = 'ABB Go To Conveyour 2'
  600 = 'ABB Go To Home'
  601 = 'ABB Go To Sensor'
  602 = 'ABB Go To Storage'
  603 = 'ABB Go To Table'
  548 = 'ABB PickLeave Conv. 1'
  549 = 'ABB PickLeave Conv. 2'
  544 = 'ABB PickLeave Sensor'
  545 = 'ABB PickLeave Storage'
  546 = 'ABB PickLeave Table'
  847 = 'ABB Status'
  562 = 'Busy'
  563 = 'Communicator'
  547 = 'Communicator Enable'
  312 = 'Done'
  315 = 'Error'
  564 = 'Error %s'
  313 = 'Executing'
  311 = 'Function call'
  61 = 'Gantry Leave'
  60 = 'Gantry Pick'
  170 = 'Heart beat'
  849 = 'Operating mode %d'
  550 = 'Pick'
  551 = 'Pos\n%s'
  63 = 'Pos \n%s'
  171 = 'Program number: %d'
  169 = 'RPC Remote Procedural Call'
  168 = 'Running'
  848 = 'Running mode %d'
  62 = 'Station\n%s'
  649 = 'Station address \n%s'
  486 = 'STN200'
  314 = 'Waiting'
END_TEXTLIST

// ---- VISUs/Visualization.TcVIS
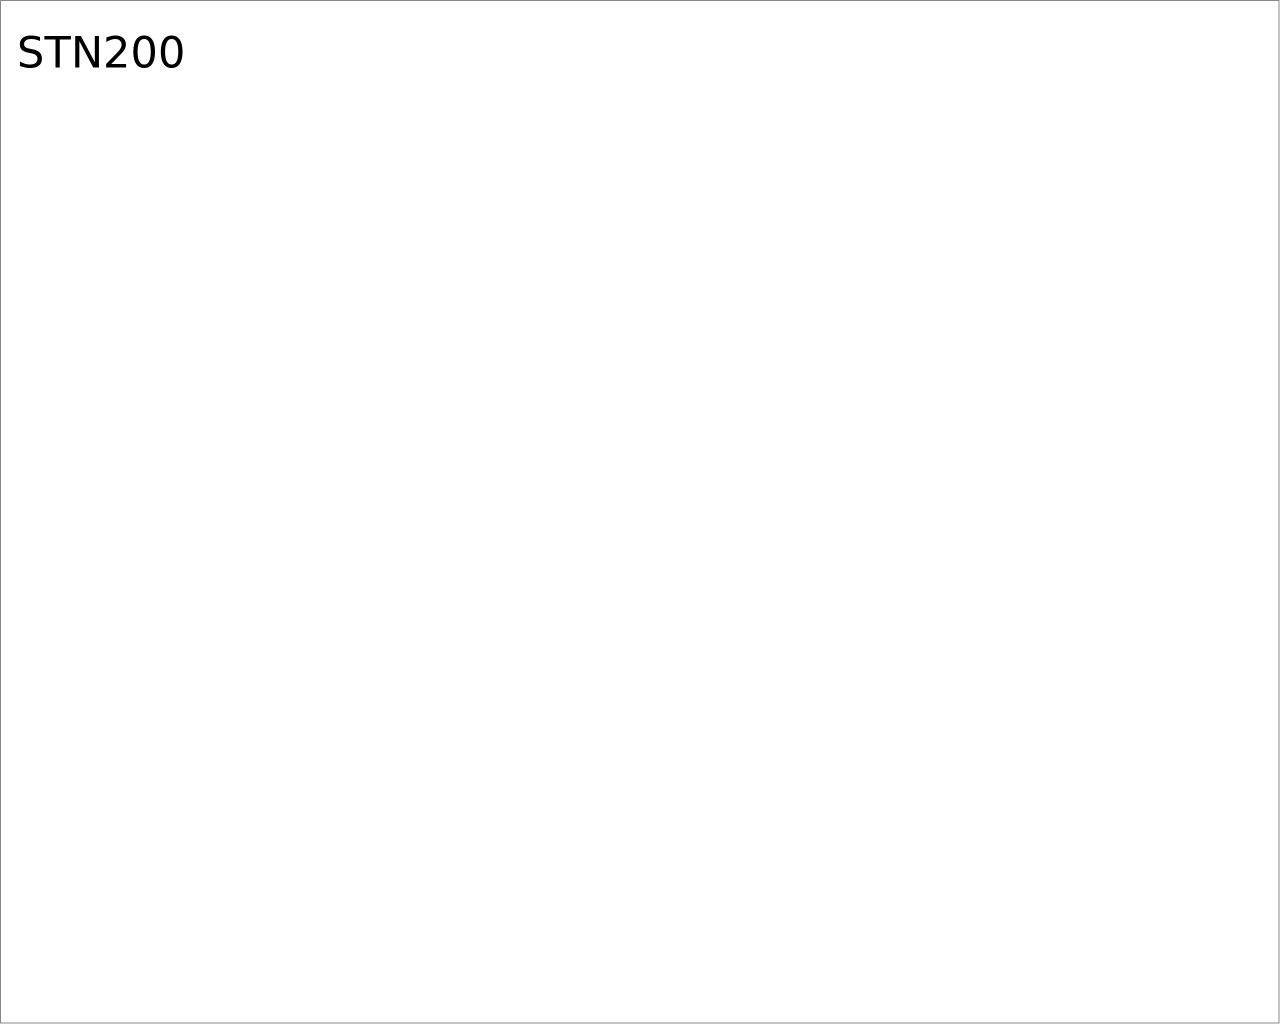
VISUALIZATION Visualization  // 1280x1024
    Label (-12,4 227x97), "STN200"
END_VISUALIZATION
